# EPICS IOC start-up script: iocsh/cav-selector.iocsh
dbLoadRecords("cav-selector.db", "P=LLRF-Ctrl:")
